// TIA Portal V17 export
// export: Created 2024-03-30T11:15:04.885183Z, ExportSetting WithDefaults, DisplayName Totally Integrated Automation Portal, DisplayVersion V17, DisplayName TIA Portal Openness, DisplayVersion V17, DisplayName TIA Portal Version Control Interface, DisplayVersion V17, DisplayName STEP 7 Professional, DisplayVersion V17, DisplayName STEP 7 Safety, DisplayVersion V17, DisplayName WinCC Advanced, DisplayVersion V17
TYPE "typ_SetupAxis"
// stored: IsFailsafeCompliant false
   STRUCT
      x_Setup_Activ : Bool;   // Set up calibration active
      i_AxisSelection : Int;   // Number of the axis
      i_Function : Int;   // 0 = automatic, 10 = ref. Travel, 20 = tap, 30 = tap with step width, 40 = start
      x_Set_Ref_Pos : Bool;   // Set reference value
      x_Set_Soft_End_Pos : Bool;   // Set software end positions
      x_Approach_Ref_Pos : Bool;   // Approach reference
      x_Axis_Pos : Bool;   // Axis positiv
      x_Axis_Neg : Bool;   // Axis negative
      x_Approach_Target_Pos : Bool;   // Approach Target position
      w_Increment : Word;   // Increments per step
      i_PWM : Int;   // PWM Signal
      di_Target_Position : DInt;   // Target position
      di_ActualPosition : DInt;   // Actual position
      di_Ref_Pos : DInt;   // Reference position
      di_Actual_Ref_Pos : DInt;   // Current reference position
      di_Soft_End_Pos_Neg : DInt;   // Software end position negative
      di_Actual_Soft_End_Pos_Neg : DInt;   // Current software end position negative
      di_Soft_End_Pos_Pos : DInt;   // Software end position positiv
      di_Actual_Soft_End_Pos_Pos : DInt;   // Current software end position positiv
      di_LoopValue : DInt;   // Loop value
   END_STRUCT;
END_TYPE
